FUNCTION_BLOCK FB_ReadHead EXTENDS FB_Base
VAR_INPUT
END_VAR
VAR_OUTPUT
END_VAR
VAR
	//eGetSource									: E_Convoyer;
	eReadDestination						: E_Convoyer;
	bExecute										: BOOL;
	fbDrand											: DRAND;
	aDestinationListe      			: ARRAY[1..4] OF UINT := [3, 6, 9, 12];
	
END_VAR

//================== Must!!
SUPER^();  
IF NOT Enable THEN RETURN; END_IF;

PROPERTY Execute : BOOL
GET
Execute := bExecute;
END_GET
SET
bExecute := Execute;
END_SET
END_PROPERTY

//FB_Init ist immer implizit verfügbar und wird primär für die Initialisierung verwendet.
//Der Rückgabewert wird nicht ausgewertet. Für gezielte Einflussnahme können Sie
//die Methoden explizit deklarieren und darin mit dem Standard-Initialisierungscode 
//zusätzlichen Code bereitstellen. Sie können den Rückgabewert auswerten.
METHOD FB_Init: BOOL
VAR_INPUT    
	bInitRetains					: BOOL; 					// TRUE: Die Retain-Variablen werden initialisiert (Reset warm / Reset kalt)    
	bInCopyCode						: BOOL;  					// TRUE: Die Instanz wird danach in den Kopiercode kopiert (Online-Change)
	
	I_Name                : STRING;         //  Name
	I_ID                  : UINT;            // ID
END_VAR
END_METHOD

METHOD mRead : E_CmdState
VAR_INPUT
	I_bExecute		: BOOL;
END_VAR

VAR
	L_uiReadData					: UINT;
	L_uiIndex							: INT;
	
END_VAR

IF NOT I_bExecute 
	THEN
    mRead := E_CmdState.Idle;
    RETURN;
END_IF

fbDrand(); 
L_uiIndex			:= LREAL_TO_INT(((fbDrand.Num) * 4)+1);
IF L_uiIndex < 1 THEN L_uiIndex := 1; END_IF;
IF L_uiIndex > 4 THEN L_uiIndex := 4; END_IF;
L_uiReadData 	:= aDestinationListe[L_uiIndex];
bExecute			:= FALSE;

CASE L_uiReadData OF
	3 : eReadDestination  := E_Convoyer.Convoyer_3;
	6 : eReadDestination 	:= E_Convoyer.Convoyer_6; 
	9 : eReadDestination 	:= E_Convoyer.Convoyer_9;
 12 : eReadDestination 	:= E_Convoyer.Convoyer_12;
ELSE
    mRead 						:= E_CmdState.Error;
    RETURN;
END_CASE

mRead := E_CmdState.Succeeded;
END_METHOD

PROPERTY ReadDestination : E_Convoyer
GET
ReadDestination := eReadDestination;
END_GET
SET
eReadDestination := ReadDestination;
END_SET
END_PROPERTY

END_FUNCTION_BLOCK

(* stored: Version 1.1.0.1, ProductVersion 3.1.4026.18
   POU FB_ReadHead: Id {7b3aad50-65da-4b94-b70d-8f823da603e1}, SpecialFunc None
   Folder 01 Properties: Id {b2440afa-7c1f-40b4-9cbc-93b18aee1299}
   Folder 02 Methodes: Id {ffaef3c6-238b-4512-a039-09cfff86c625}
   Property Execute: Id {c4f10ddb-f559-40f1-8458-77d837f34033}
   Get Get: Id {43609412-b8d4-4ece-84fb-c6e1262b1d19}
   Set Set: Id {83f95d42-f479-48cd-a74e-49b2984b823f}
   Method FB_Init: Id {e8a7e786-1a56-4f8b-9239-87a55b695227}
   Method mRead: Id {f10879c1-6084-4c42-b497-6acc39e492c3}
   Property ReadDestination: Id {1ddf43fd-fbf7-481e-a044-6c3e0841a14e}
   Get Get: Id {180394fd-6b2f-4234-94af-956eac736f2f}
   Set Set: Id {9605183d-64b3-424c-af0f-e291f6b3fa2e} *)
